{attribute 'no_explicit_call' := 'Body contains no logic, calling methods only allowed.'}
PROGRAM JXCE1_Helper
VAR
END_VAR

// Returns the controller state based on various signals of the controller
METHOD GetControllerState	: E_JXCE1_State
VAR_INPUT
	controller	: I_JXCE1_StepperMotorControl;
END_VAR
IF  NOT controller.Status.Busy AND
	NOT controller.Status.Done AND
	NOT controller.Status.MotorOn AND
	NOT controller.Status.SETON AND
	controller.Status.StepData = 0 
THEN
	GetControllerState := E_JXCE1_State.POWER_OFF;
	RETURN;
END_IF

IF  NOT controller.Status.Busy AND
	NOT controller.Status.Done AND
	controller.Status.MotorOn AND
	NOT controller.Status.SETON AND
	controller.Status.StepData = 0 
THEN
	GetControllerState := E_JXCE1_State.POWER_ON_NO_MOTION;
	RETURN;
END_IF

IF  controller.Status.Busy AND
	NOT controller.Status.Done AND
	controller.Status.MotorOn AND
	NOT controller.Status.SETON AND
	controller.Status.StepData = 0 
THEN
	GetControllerState := E_JXCE1_State.RETURNING_TO_ORIGIN;
	RETURN;
END_IF

IF  NOT controller.Status.Busy AND
	controller.Status.Done AND
	controller.Status.MotorOn AND
	controller.Status.SETON AND
	controller.Status.StepData = 0 
THEN
	GetControllerState := E_JXCE1_State.AT_ORIGIN_POSITION;
	RETURN;
END_IF

IF  controller.Status.Busy AND
	NOT controller.Status.Done AND
	controller.Status.MotorOn AND
	controller.Status.SETON AND
	controller.Status.StepData <> 0 {warning 'preveri, ne vem vrednosti...'}
THEN
	GetControllerState := E_JXCE1_State.POSITIONING_OR_PUSHING_ACTIVE;
	RETURN;
END_IF

IF  NOT controller.Status.Busy AND
	NOT controller.Status.Done AND
	controller.Status.MotorOn AND
	controller.Status.SETON AND
	controller.Status.StepData <> 0 {warning 'preveri, ne vem vrednosti...'}
THEN
	GetControllerState := E_JXCE1_State.HOLD;
	RETURN;
END_IF

IF  NOT controller.Status.Busy AND
	controller.Status.Done AND
	controller.Status.MotorOn AND
	controller.Status.SETON AND
	controller.Status.StepData <> 0 {warning 'preveri, ne vem vrednosti...'}
THEN
	GetControllerState := E_JXCE1_State.POSITIONING_COMPLETE;
	RETURN;
END_IF

IF  NOT controller.Status.Busy AND
	controller.Status.Done AND
	controller.Status.MotorOn AND
	controller.Status.SETON AND
	controller.Status.StepData <> 0 {warning 'preveri, ne vem vrednosti...'}
THEN
	GetControllerState := E_JXCE1_State.PUSHING_COMPLETED;
	RETURN;
END_IF

IF  NOT controller.Status.Busy AND
	NOT controller.Status.Done AND
	controller.Status.MotorOn AND
	controller.Status.SETON AND
	controller.Status.StepData = 0
THEN
	GetControllerState := E_JXCE1_State.PUSHING_STOPPED_NO_WORKLOAD_DETECTED;
	RETURN;
END_IF

IF  NOT controller.Status.Busy AND
	NOT controller.Status.Done AND
	NOT controller.Status.MotorOn AND
	controller.Status.SETON AND
	controller.Status.StepData <> 0 {warning 'preveri, ne vem vrednosti...'}
THEN
	GetControllerState := E_JXCE1_State.SERVO_OFF_AFTER_RETURNING_TO_ORIGIN;
	RETURN;
END_IF

IF  NOT controller.Status.Busy AND
	NOT controller.Status.Done AND
	NOT controller.Status.MotorOn AND
	controller.Status.SETON AND
	controller.Status.StepData = 0
THEN
	GetControllerState := E_JXCE1_State.EMERGENCY;
	RETURN;
END_IF
END_METHOD

END_PROGRAM

(* stored: Version 1.1.0.1, ProductVersion 3.1.4024.15
   POU JXCE1_Helper: Id {7943e6f3-dd33-436c-a4de-3f4a51de3c7b}, SpecialFunc None
   Method GetControllerState: Id {b0528bb9-d3a1-4c2b-a4fa-fbe6d6ccfde8} *)
